FUNCTION_BLOCK FB_CommandChangeStart EXTENDS FB_CommandChange IMPLEMENTS ITF_CommandChange
VAR

END_VAR

METHOD Execute : BOOL
VAR_INPUT
END_VAR
END_METHOD

METHOD FB_init : BOOL
VAR_INPUT
	bInitRetains : BOOL; // if TRUE, the retain variables are initialized (warm start / cold start)
	bInCopyCode : BOOL;  // if TRUE, the instance afterwards gets moved into the copy code (online change)
END_VAR
THIS^.SetText (eLocation := E_BaseLocation.pl, wsDescription := "Command change state - Start");
THIS^.SetText (eLocation := E_BaseLocation.en, wsDescription := "Command change state - Start");
THIS^.SetText (eLocation := E_BaseLocation.de, wsDescription := "Command change state - Start");
THIS^.SetName (stName := THIS^.GetTexts ());
END_METHOD

END_FUNCTION_BLOCK

(* stored: Version 1.1.0.1
   POU FB_CommandChangeStart: Id {3e97eb6b-0aae-0d44-3f5a-d06acc717999}, SpecialFunc None
   Method Execute: Id {61a00f7e-77a7-075e-3e41-e4b391a63760}
   Method FB_init: Id {8a8b6ee8-32b2-028a-07da-958bf1cc3ceb} *)
